// TwinCAT 3 PLC project MPLR
// ProgramVersion: 3.1.4026.19
// libraries:
//   Tc2_MC2, * (Beckhoff Automation GmbH)
//   Tc2_SerialCom, * (Beckhoff Automation GmbH)
//   Tc2_Standard, * (Beckhoff Automation GmbH)
//   Tc2_System, * (Beckhoff Automation GmbH)
//   Tc2_Utilities, * (Beckhoff Automation GmbH)
//   Tc3_Vision, * (Beckhoff Automation GmbH)
//   Tc3_Weighing, * (Beckhoff Automation GmbH)
// project tree:
//   DUTs/ E_PlateNum.TcDUT, MoveState_t.TcDUT, ST_CameraControl.TcDUT, ST_Origins.TcDUT, ST_PoseLREAL.TcDUT, ST_StepperMotorControl.TcDUT, ST_Transitions.TcDUT
//   DUTs/Robot/ur_input/ UR_1_T2O_Robot.TcDUT, UR_1_T2O_Safety.TcDUT, UR_1_T2O_State.TcDUT, UR_2_T2O_IO.TcDUT, UR_2_T2O_IOs.TcDUT, UR_2_T2O_Tool.TcDUT, UR_3_T2O_Joints.TcDUT, UR_4_T2O_TCP.TcDUT, UR_5_T2O_BitRegisters.TcDUT, UR_6_T2O_IntRegisters.TcDUT, UR_7_T2O_FloatRegisters.TcDUT, UR_T2O.TcDUT
//   DUTs/Robot/ur_output/ UR_8_O2T_IOs.TcDUT, UR_8_O2T_Robot.TcDUT, UR_8_O2T_Robot_IO.TcDUT, UR_9_O2T_Bits1.TcDUT, UR_9_O2T_Bits2.TcDUT, UR_9_O2T_Floats.TcDUT, UR_9_O2T_Ints.TcDUT, UR_9_O2T_Registers1.TcDUT, UR_9_O2T_Registers2.TcDUT, UR_O2T.TcDUT
//   GVLs/ process_gvl.TcGVL
//   / PlcTask.TcTTO
//   POUs/ FB_CreateTransformationMat.TcPOU, FB_LoadCell.TcPOU, FB_MagStirrer.TcPOU, FB_MatConversion.TcPOU, FB_MotorJog.TcPOU, FB_MultiplyMatrices4x4.TcPOU, FB_PeristalticPump.TcPOU, FB_Robot.TcPOU, FB_Camera.TcPOU, FB_SerialCom.TcPOU, FB_Test.TcPOU, MAIN.TcPOU, MPLR_UML.TcCD (not stored)
//   POUs/Modules/ FB_LoadingStationA.TcPOU, FB_SolidSamplingModule.TcPOU, FB_StirringModule.TcPOU
// real-time tasks:
//   TASK PlcTask: cycle T#10ms, priority 20, ADS port 350
//   TASK VnTask ImgAcq (Camera Daheng): cycle T#1ms, priority 5, ADS port 351
//   TASK VnTask ADS (Camera Daheng): cycle T#10ms, priority 6, ADS port 352
//   TASK VnTask ImgAcq (Daheng): cycle T#1ms, priority 7, ADS port 353
//   TASK VnTask ADS (Daheng): cycle T#10ms, priority 8, ADS port 354
//   TASK RTTask: cycle T#1ms, priority 1, ADS port 301
// motion (NC):
//   TASK NC-Task 1 SAF: cycle T#2ms, priority 4, ADS port 501
//   TASK NC-Task 1 SVB: cycle T#10ms, priority 9, ADS port 511
//   AXIS Axis 2 (id 2)
//     Dynamic: Acceleration=1314.17, Deceleration=1314.17, Jerk=3942.52
//     Velo: RefSearch=8.76116, RefSync=8.76116, SlowManual=43.8058, FastManual=262.8348, Fast=876.116, Maximum=876.116
//     PositionAreaControl: Enable=false
//     TargetPosControl: Enable=false
//     OtherSettings: AllowMotionCmdToSlave=true
//     encoder EncType=19
//       EncPara: ScaleFactorNumerator=60, ScaleFactorDenominator=1048576, MaxCount=#xffffffff
//         SoftEndMinControl: Range=5
//         SoftEndMaxControl: Range=17
//     drive DrvType=16
//       DrvPara: MaxCount=#xffffffff, DriveControlDWord=#x00020100
//         Analog: VeloReferenz=963.7276, VeloScale=32, TorqueSetpointScale=10, ScaleFactorActTorque=0.1
//         TimeComp: TaskDelayCycles=1
//     controller CtrType=1
//       CtrPara: PriorControlFactor=1
//         PosDiffControl: Enable=false
//         Observer: BandWidth=20
// I/O:
//   DEVICE Device 1 (EtherCAT), AmsNetId 5.146.234.225.2.1
//     Term 7 (EK1200) [EK1200-5000 EtherCAT Power supply (2A E-Bus)]
//       Term 7 (EL7062) [EL7062-0000 2Ch. Stepper motor output stage (48V, 3A)]
//         startup 32785:27 := 6C030000 // DRV Motor Settings Ch.1 / Motor speed limitation
//         startup 28688:3 := 08 // DRV Outputs Ch.1 / Modes of operation
//         startup 28688:16 := FF7F // DRV Outputs Ch.1 / Positive torque limit value
//         startup 28688:17 := FF7F // DRV Outputs Ch.1 / Negative torque limit value
//         startup 32784:87 := 64 // DRV Amplifier Settings Ch.1 / Position loop velocity feed forward gain
//         startup 32784:109 := 64000000 // DRV Amplifier Settings Ch.1 / Torque feed forward gain
//         startup 32785:52 := 70170000 // DRV Motor Settings Ch.1 / Configured motor current
//         startup 32784:19 := 1D00 // DRV Amplifier Settings Ch.1 / Current loop proportional gain
//         startup 32784:18 := 1E00 // DRV Amplifier Settings Ch.1 / Current loop integral time
//         startup 32784:21 := 91000000 // DRV Amplifier Settings Ch.1 / Velocity loop proportional gain
//         startup 32784:20 := 96000000 // DRV Amplifier Settings Ch.1 / Velocity loop integral time
//         startup 32776:18 := 0100 // FB Settings ENC Ch.1 / Encoder type
//         startup 32784:100 := 12 // DRV Amplifier Settings Ch.1 / Commutation type
//       Term 3 (EL1008) [EL1008 8Ch. Dig. Input 24V, 3ms]
//       Term 4 (EL3078) [EL3078 8Ch. Ana. Input +/-10V, +/-20mA]
//       Term 5 (EL2008) [EL2008 8Ch. Dig. Output 24V, 0.5A]
//       Term 12 (EL6002) [EL6002 Interface 2Ch. (RS232)]
//       Term 13 (EL9011) [EL9011 End Terminal]
//   DEVICE Device 3 (RT-Ethernet Adapter)
//   DEVICE Device 2 (Profinet Controller), AmsNetId 5.146.234.225.3.1
//     uriodev1 [Universal Robots A/S UR IO device, for PNIO controller with PDev 0000201]
//       modules: Term 1 (DAP Module), Term 2 (1_T2O State), Term 3 (2_T2O IO), Term 4 (3_T2O Joints), Term 5 (4_T2O TCP), Term 6 (5_T2O General Purpose Bit Registers), Term 7 (6_T2O General Purpose Int Registers), Term 8 (7_T2O General Purpose Float Registers), Term 9 (8_O2T Robot IO), Term 10 (9_O2T General Purpose Registers 1), Term 11 (10_O2T General Purpose Registers 2)
// variable links:
//   NC-Task 1 SAF/Axes/Axis 2 <-> Device 1 (EtherCAT)/Term 7 (EK1200)/Term 7 (EL7062)
//     Drive/Inputs/In/nDataIn1 <-> DRV Following error actual value Channel 1/Following error actual value
//     Drive/Inputs/In/nDcOutputTime <-> InfoData/DcOutputShift
//     Drive/Inputs/In/nState1 <-> DRV Statusword Channel 1/Statusword
//     Drive/Inputs/In/nState2 <-> DRV Statusword Channel 1/Statusword @bit 8
//     Drive/Inputs/In/nState4 @bit 1 <-> WcState/InputToggle
//     Drive/Inputs/In/nState4 <-> WcState/WcState
//     Drive/Outputs/Out/nCtrl1 <-> DRV Controlword Channel 1/Controlword
//     Drive/Outputs/Out/nCtrl2 <-> DRV Controlword Channel 1/Controlword @bit 8
//     Drive/Outputs/Out/nDataOut1 <-> DRV Target position Channel 1/Target position
//     Enc/Inputs/In/nDataIn1 <-> FB Position Channel 1/Position
//     Enc/Inputs/In/nDcInputTime <-> InfoData/DcInputShift
//     Enc/Inputs/In/nState4 @bit 1 <-> WcState/InputToggle
//     Enc/Inputs/In/nState4 <-> WcState/WcState
//   mplr/mplr Instance <-> Device 2 (Profinet Controller)/uriodev1
//     PlcTask Inputs/process_gvl.fRobotInput/General_Bits <-> API/Term 6 (5_T2O General Purpose Bit Registers)/Subterm 8 (5_T2O General Purpose Bit Registers)/Inputs/T2O Bit Registers
//     PlcTask Inputs/process_gvl.fRobotInput/General_Float/Floats <-> API/Term 8 (7_T2O General Purpose Float Registers)/Subterm 10 (7_T2O General Purpose Float Registers)/Inputs/T2O Float Registers
//     PlcTask Inputs/process_gvl.fRobotInput/General_Int/Ints <-> API/Term 7 (6_T2O General Purpose Int Registers)/Subterm 9 (6_T2O General Purpose Int Registers)/Inputs/T2O Int Registers
//     PlcTask Inputs/process_gvl.fRobotInput/IO <-> API/Term 3 (2_T2O IO)/Subterm 5 (2_T2O IO)/Inputs/T2O IO
//     PlcTask Inputs/process_gvl.fRobotInput/Joints <-> API/Term 4 (3_T2O Joints)/Subterm 6 (3_T2O Joints)/Inputs/T2O Joints
//     PlcTask Inputs/process_gvl.fRobotInput/State <-> API/Term 2 (1_T2O State)/Subterm 4 (1_T2O State)/Inputs/T2O State
//     PlcTask Inputs/process_gvl.fRobotInput/TCP <-> API/Term 5 (4_T2O TCP)/Subterm 7 (4_T2O TCP)/Inputs/T2O TCP
//     PlcTask Outputs/process_gvl.fRobotOutput/General_Register1 <-> API/Term 10 (9_O2T General Purpose Registers 1)/Subterm 12 (9_O2T General Purpose Registers 1)/Outputs/O2T Reg 1
//     PlcTask Outputs/process_gvl.fRobotOutput/General_Register2 <-> API/Term 11 (10_O2T General Purpose Registers 2)/Subterm 13 (10_O2T General Purpose Registers 2)/Outputs/O2T Reg 2
//     PlcTask Outputs/process_gvl.fRobotOutput/IO <-> API/Term 9 (8_O2T Robot IO)/Subterm 11 (8_O2T Robot IO)/Outputs/O2T IO
//   mplr/mplr Instance <-> NC-Task 1 SAF/Axes/Axis 2
//     PlcTask Inputs/MAIN.fbMotorJog.Axis1.NcToPlc <-> Outputs/ToPlc
//     PlcTask Outputs/MAIN.fbMotorJog.Axis1.PlcToNc <-> Inputs/FromPlc

CONFIGURATION MPLR
    RESOURCE PLC ON TwinCAT3
        TASK PlcTask(INTERVAL := T#10ms, PRIORITY := 20);
        PROGRAM MAIN WITH PlcTask : MAIN;
    END_RESOURCE
END_CONFIGURATION

// ---- DUTs/E_PlateNum.TcDUT
{attribute 'qualified_only'}
{attribute 'strict'}
{attribute 'to_string'}
TYPE E_PlateNum :
(
	ePlate1 := 0,
	ePlate2,
	ePlate3,
	ePlate4,
	ePlate5,
	ePlate6,
	ePlate7,
	ePlate8
);
END_TYPE

// ---- DUTs/MoveState_t.TcDUT
// {attribute 'qualified_only'}
// {attribute 'strict'}
// {attribute 'to_string'}
TYPE MoveState_t :
(
	MOVESTATE_INIT,
	MOVESTATE_ENABLE,
	MOVESTATE_IDLE,
	MOVESTATE_FORWARD,
	MOVESTATE_BACKWARDS,
	MOVESTATE_HALT,
	MOVESTATE_BACKWARDSSLOW,
	MOVESTATE_NEWTARGETPOSITION,
	MOVESTATE_ERROR,
	MOVESTATE_RESET
) UDINT;
END_TYPE

// ---- DUTs/Robot/ur_input/UR_1_T2O_Robot.TcDUT
TYPE UR_1_T2O_Robot :
STRUCT
	Controller_major_version:USINT;
	Controller_minor_version:USINT;
	Reserved:UInt;
	Robot_mode:USInt;
	Real_time_machine_seconds:USInt;
	Real_time_machine_milliseconds:UInt;
	Real_time_machine_minutes:USInt;
	Real_time_machine_hours:USInt;
	Real_time_machine_days:UINT;
	Robot_current_A:REAL;
	Is_power_on:BIT;
	Is_program_running:BIT;
	Is_teach_button_pressed:BIT;
	Is_power_button_pressed:BIT;
	Reserved_4:BIT;
	Reserved_5:BIT;
	Reserved_6:BIT;
	Reserved_7:BIT;
	Reserved_8_15:USInt;
	Reserved_16_31:UINT;
	Speed_slider_fraction:REAL;
END_STRUCT
END_TYPE

// ---- DUTs/Robot/ur_input/UR_1_T2O_Safety.TcDUT
TYPE UR_1_T2O_Safety :
STRUCT
	Safety_mode:USINT;
	Reserved_1:USINT;
	Reserved_2:UInt;
	Is_normal_mode:BIT;
	Is_reduced_mode:BIT;
	Is_protective_stopped:BIT;
	Is_recovery_mode:BIT;
	Is_safeguard_stopped:BIT;
	Is_system_emergency_stopped:BIT;
	Is_robot_emergency_stopped:BIT;
	Is_emergency_stopped:BIT;
	Is_violation:BIT;
	Is_fault:BIT;
	Is_stopped_due_to_safety:BIT;
	Reserved_11:BIT;
	Reserved_12:BIT;
	Reserved_13:BIT;
	Reserved_14:BIT;
	Reserved_15:BIT;
	Reserved_16_31:UINT;
END_STRUCT
END_TYPE

// ---- DUTs/Robot/ur_input/UR_1_T2O_State.TcDUT
TYPE UR_1_T2O_State :
STRUCT
      Robot : UR_1_T2O_Robot;
      Safety : UR_1_T2O_Safety;
END_STRUCT
END_TYPE

// ---- DUTs/Robot/ur_input/UR_2_T2O_IO.TcDUT
TYPE UR_2_T2O_IO :
STRUCT
	  IOs : UR_2_T2O_IOs;
	  Tool : UR_2_T2O_Tool;
END_STRUCT
END_TYPE

// ---- DUTs/Robot/ur_input/UR_2_T2O_IOs.TcDUT
TYPE UR_2_T2O_IOs :
STRUCT
	Standard_digital_inputs : USINT;
	Configurable_digital_inputs:USINT;
	Standard_digital_outputs:USINT;
	Configurable_digital_outputs:USINT;
	Analog_IO_types:USINT;
	Reserved_8_15:USINT;
	Reserved_16_31:UINT;
	Standard_analog_input_A_or_V:ARRAY[0..1] OF REAL;
	Standard_analog_output_A_or_V:ARRAY[0..1] OF REAL;
	IO_current_A:REAL;
	Euromap67_input_bits:ARRAY[0..3] OF BYTE;
	Euromap67_output_bits:ARRAY[0..3] OF BYTE;
	Euromap67_24V_voltage:REAL;
	Euromap67_24V_current:REAL;
END_STRUCT
END_TYPE

// ---- DUTs/Robot/ur_input/UR_2_T2O_Tool.TcDUT
TYPE UR_2_T2O_Tool :
STRUCT
	Tool_mode:USINT;
	Reserved_7_15:USINT;
	Reserved_16_31:UINT;
	Tool_Digital_Inputs:USINT;
	Tool_Digital_Outputs:USINT;
	Tool_Analog_Input_Types:USINT;
	Reserved_24_31:USINT;
	Tool_analog_input_A_OR_V:ARRAY[0..1] OF REAL;
	Tool_output_voltage_V:REAL;
	Tool_current_A:REAL;
END_STRUCT
END_TYPE

// ---- DUTs/Robot/ur_input/UR_3_T2O_Joints.TcDUT
TYPE UR_3_T2O_Joints :
STRUCT
	Joint_position_rad:ARRAY[0..5] OF REAL;
	Joint_velocity_radS:ARRAY[0..5] OF REAL;
	Joint_current_A:ARRAY[0..5] OF REAL;
	Joint_temperature_C:ARRAY[0..5] OF REAL;
	Joint_mode:ARRAY[0..5] OF USINT;
	Reserved_9:UINT;
END_STRUCT
END_TYPE

// ---- DUTs/Robot/ur_input/UR_4_T2O_TCP.TcDUT
TYPE UR_4_T2O_TCP :
STRUCT
	TCP_Position_XYZ_m:ARRAY[0..2] OF REAL;
	TCP_Position_RXRYRZ_rad:ARRAY[0..2] OF REAL;
	TCP_velocity_XYZ_m_S:ARRAY[0..2] OF REAL;
	TCP_velocity_RXRYRZ_rad_S:ARRAY[0..2] OF REAL;
	TCP_force_XYZ_N:ARRAY[0..2] OF REAL;
	TCP_torque_XYZ_Nm:ARRAY[0..2] OF REAL;
	TCP_force_scalar_N:REAL;
END_STRUCT
END_TYPE

// ---- DUTs/Robot/ur_input/UR_5_T2O_BitRegisters.TcDUT
TYPE UR_5_T2O_BitRegisters :
STRUCT
	GPBitIN_0 : BIT;
	GPBitIN_1 : BIT;
	GPBitIN_2 : BIT;
	GPBitIN_3 : BIT;
	GPBitIN_4 : BIT;
	GPBitIN_5 : BIT;
	GPBitIN_6 : BIT;
	GPBitIN_7 : BIT;
	GPBitIN_8 : BIT;
	GPBitIN_9 : BIT;
	GPBitIN_10 : BIT;
	GPBitIN_11 : BIT;
	GPBitIN_12 : BIT;
	GPBitIN_13 : BIT;
	GPBitIN_14 : BIT;
	GPBitIN_15 : BIT;
	GPBitIN_16 : BIT;
	GPBitIN_17 : BIT;
	GPBitIN_18 : BIT;
	GPBitIN_19 : BIT;
	GPBitIN_20 : BIT;
	GPBitIN_21 : BIT;
	GPBitIN_22 : BIT;
	GPBitIN_23 : BIT;
	GPBitIN_24 : BIT;
	GPBitIN_25 : BIT;
	GPBitIN_26 : BIT;
	GPBitIN_27 : BIT;
	GPBitIN_28 : BIT;
	GPBitIN_29 : BIT;
	GPBitIN_30 : BIT;
	GPBitIN_31 : BIT;
	GPBitIN_32 : BIT;
	GPBitIN_33 : BIT;
	GPBitIN_34 : BIT;
	GPBitIN_35 : BIT;
	GPBitIN_36 : BIT;
	GPBitIN_37 : BIT;
	GPBitIN_38 : BIT;
	GPBitIN_39 : BIT;
	GPBitIN_40 : BIT;
	GPBitIN_41 : BIT;
	GPBitIN_42 : BIT;
	GPBitIN_43 : BIT;
	GPBitIN_44 : BIT;
	GPBitIN_45 : BIT;
	GPBitIN_46 : BIT;
	GPBitIN_47 : BIT;
	GPBitIN_48 : BIT;
	GPBitIN_49 : BIT;
	GPBitIN_50 : BIT;
	GPBitIN_51 : BIT;
	GPBitIN_52 : BIT;
	GPBitIN_53 : BIT;
	GPBitIN_54 : BIT;
	GPBitIN_55 : BIT;
	GPBitIN_56 : BIT;
	GPBitIN_57 : BIT;
	GPBitIN_58 : BIT;
	GPBitIN_59 : BIT;
	GPBitIN_60 : BIT;
	GPBitIN_61 : BIT;
	GPBitIN_62 : BIT;
	GPBitIN_63 : BIT;
END_STRUCT
END_TYPE

// ---- DUTs/Robot/ur_input/UR_6_T2O_IntRegisters.TcDUT
TYPE UR_6_T2O_IntRegisters :
STRUCT
		Ints:ARRAY[0..23] OF DINT;
END_STRUCT
END_TYPE

// ---- DUTs/Robot/ur_input/UR_7_T2O_FloatRegisters.TcDUT
TYPE UR_7_T2O_FloatRegisters :
STRUCT
	  Floats : ARRAY[0..23] OF REAL;
END_STRUCT
END_TYPE

// ---- DUTs/Robot/ur_input/UR_T2O.TcDUT
TYPE UR_T2O :
STRUCT
	State:UR_1_T2O_State;
	IO:UR_2_T2O_IO;
	Joints:UR_3_T2O_Joints;
	TCP:UR_4_T2O_TCP;
	General_Bits:UR_5_T2O_BitRegisters;
	General_Int:UR_6_T2O_IntRegisters;
	General_Float:UR_7_T2O_FloatRegisters;
END_STRUCT
END_TYPE

// ---- DUTs/Robot/ur_output/UR_8_O2T_IOs.TcDUT
TYPE UR_8_O2T_IOs :
STRUCT
	Standard_digital_output_mask:USINT;
	Configurable_digital_output_mask:USINT;
	Standard_digital_outputs:USINT;
	Configurable_digital_outputs:USINT;
	Analog_output_mask:USINT;
	Analog_output_types:USINT;
	Tool_digital_output_mask:USINT;
	Tool_digital_output:USINT;
	Standard_analog_output:ARRAY[0..1] OF REAL;
END_STRUCT
END_TYPE

// ---- DUTs/Robot/ur_output/UR_8_O2T_Robot.TcDUT
TYPE UR_8_O2T_Robot :
STRUCT
	  Speed_slider_fraction_mask : BIT;
	  Reserved_1 : BIT;
	  Reserved_2 : BIT;
	  Reserved_3 : BIT;
	  Reserved_4 : BIT;
	  Reserved_5 : BIT;
	  Reserved_6 : BIT;
	  Reserved_7 : BIT;
	  Reserved_8_15 : USINT;
	  Reserved_16_31 : UINT;
	  Speed_slider_fraction : REAL;
END_STRUCT
END_TYPE

// ---- DUTs/Robot/ur_output/UR_8_O2T_Robot_IO.TcDUT
TYPE UR_8_O2T_Robot_IO :
STRUCT
      Robot : UR_8_O2T_Robot;
      IOs : UR_8_O2T_IOs;
END_STRUCT
END_TYPE

// ---- DUTs/Robot/ur_output/UR_9_O2T_Bits1.TcDUT
TYPE UR_9_O2T_Bits1 :
STRUCT
	GPBitIN_0 : BIT;
	GPBitIN_1 : BIT;
	GPBitIN_2 : BIT;
	GPBitIN_3 : BIT;
	GPBitIN_4 : BIT;
	GPBitIN_5 : BIT;
	GPBitIN_6 : BIT;
	GPBitIN_7 : BIT;
	GPBitIN_8 : BIT;
	GPBitIN_9 : BIT;
	GPBitIN_10 : BIT;
	GPBitIN_11 : BIT;
	GPBitIN_12 : BIT;
	GPBitIN_13 : BIT;
	GPBitIN_14 : BIT;
	GPBitIN_15 : BIT;
	GPBitIN_16 : BIT;
	GPBitIN_17 : BIT;
	GPBitIN_18 : BIT;
	GPBitIN_19 : BIT;
	GPBitIN_20 : BIT;
	GPBitIN_21 : BIT;
	GPBitIN_22 : BIT;
	GPBitIN_23 : BIT;
	GPBitIN_24 : BIT;
	GPBitIN_25 : BIT;
	GPBitIN_26 : BIT;
	GPBitIN_27 : BIT;
	GPBitIN_28 : BIT;
	GPBitIN_29 : BIT;
	GPBitIN_30 : BIT;
	GPBitIN_31 : BIT;
END_STRUCT
END_TYPE

// ---- DUTs/Robot/ur_output/UR_9_O2T_Bits2.TcDUT
TYPE UR_9_O2T_Bits2 :
STRUCT
	GPBitIN_32 : BIT;
	GPBitIN_33 : BIT;
	GPBitIN_34 : BIT;
	GPBitIN_35 : BIT;
	GPBitIN_36 : BIT;
	GPBitIN_37 : BIT;
	GPBitIN_38 : BIT;
	GPBitIN_39 : BIT;
	GPBitIN_40 : BIT;
	GPBitIN_41 : BIT;
	GPBitIN_42 : BIT;
	GPBitIN_43 : BIT;
	GPBitIN_44 : BIT;
	GPBitIN_45 : BIT;
	GPBitIN_46 : BIT;
	GPBitIN_47 : BIT;
	GPBitIN_48 : BIT;
	GPBitIN_49 : BIT;
	GPBitIN_50 : BIT;
	GPBitIN_51 : BIT;
	GPBitIN_52 : BIT;
	GPBitIN_53 : BIT;
	GPBitIN_54 : BIT;
	GPBitIN_55 : BIT;
	GPBitIN_56 : BIT;
	GPBitIN_57 : BIT;
	GPBitIN_58 : BIT;
	GPBitIN_59 : BIT;
	GPBitIN_60 : BIT;
	GPBitIN_61 : BIT;
	GPBitIN_62 : BIT;
	GPBitIN_63 : BIT;
END_STRUCT
END_TYPE

// ---- DUTs/Robot/ur_output/UR_9_O2T_Floats.TcDUT
TYPE UR_9_O2T_Floats :
STRUCT
	Floats : ARRAY[0..11] OF REAL;
END_STRUCT
END_TYPE

// ---- DUTs/Robot/ur_output/UR_9_O2T_Ints.TcDUT
TYPE UR_9_O2T_Ints :
STRUCT
      Ints : ARRAY[0..11] OF DINT;
END_STRUCT
END_TYPE

// ---- DUTs/Robot/ur_output/UR_9_O2T_Registers1.TcDUT
TYPE UR_9_O2T_Registers1 :
STRUCT
      Bits : UR_9_O2T_Bits1;
      Ints : UR_9_O2T_Ints;
      Floats : UR_9_O2T_Floats;
END_STRUCT
END_TYPE

// ---- DUTs/Robot/ur_output/UR_9_O2T_Registers2.TcDUT
TYPE UR_9_O2T_Registers2 :
STRUCT
      Bits : UR_9_O2T_Bits2;
      Ints : UR_9_O2T_Ints;
      Floats : UR_9_O2T_Floats;
END_STRUCT
END_TYPE

// ---- DUTs/Robot/ur_output/UR_O2T.TcDUT
TYPE UR_O2T :
STRUCT
	IO:UR_8_O2T_Robot_IO;
	General_Register1:UR_9_O2T_Registers1;
	General_Register2:UR_9_O2T_Registers1;
END_STRUCT
END_TYPE

// ---- DUTs/ST_CameraControl.TcDUT
TYPE ST_CameraControl :
STRUCT

END_STRUCT
END_TYPE

// ---- DUTs/ST_Origins.TcDUT
TYPE ST_Origins :
STRUCT
	fOrigin1		: ARRAY[0..5]	OF LREAL := [0.0, 0.0, 0.0, 0.0, 0.0, 0.0];
	fOrigin2		: ARRAY[0..5]	OF LREAL := [0.0, 0.0, 0.0, 0.0, 0.0, 0.0];
	fOrigin3		: ARRAY[0..5]	OF LREAL := [0.0, 0.0, 0.0, 0.0, 0.0, 0.0];
	fOrigin4		: ARRAY[0..5]	OF LREAL := [0.0, 0.0, 0.0, 0.0, 0.0, 0.0];
	fOrigin5		: ARRAY[0..5]	OF LREAL := [0.0, 0.0, 0.0, 0.0, 0.0, 0.0];
	fOrigin6		: ARRAY[0..5]	OF LREAL := [0.0, 0.0, 0.0, 0.0, 0.0, 0.0];
	fOrigin7		: ARRAY[0..5]	OF LREAL := [0.0, 0.0, 0.0, 0.0, 0.0, 0.0];
	fOrigin8		: ARRAY[0..5]	OF LREAL := [0.0, 0.0, 0.0, 0.0, 0.0, 0.0];
END_STRUCT
END_TYPE

// ---- DUTs/ST_PoseLREAL.TcDUT
TYPE ST_PoseLREAL :
STRUCT
	R_Mat : TcVnMatrix3x3_LREAL;
    T_Mat : TcVnVector3_LREAL;
	X_Mat : TcVnMatrix;
END_STRUCT
END_TYPE

// ---- DUTs/ST_StepperMotorControl.TcDUT
TYPE ST_StepperMotorControl :
STRUCT
// 	Axis1:AXIS_REF;
// 	MC_Power: MC_Power;
// 	MC_MoveAbsolute: MC_MoveAbsolute;
// 	bMove: BOOL;
// 	bInput AT%I*:BOOL;
// 	bEnable: BOOL;
// 	
// 	bLoadingPosition		:LREAL	:=68;
// 	bLoadingVelocity		:LREAL	:=0.5;
// 	bLoadingAcceleration	:LREAL	:=1;
// 	bLoadingDeceleration	:LREAL	:=1;
// 	
// 	bDosingPosition		:LREAL	:=64;
// 	bDosingVelocity		:LREAL	:=0.5;
// 	bDosingAcceleration	:LREAL	:=1;
// 	bDosingDeceleration	:LREAL	:=1;
END_STRUCT
END_TYPE

// ---- DUTs/ST_Transitions.TcDUT
TYPE ST_Transitions :
STRUCT
	ModulesDetected				: BOOL;
	FlaskPicked					: BOOL;
	FlaskPlaced					: BOOL;
	FingerAGripped				: BOOL;
	FingerBGripped				: BOOL;
	FingerCGripped				: BOOL;
	FingerDGripped				: BOOL;
	FingerADeGripped			: BOOL;
	FingerBDeGripped			: BOOL;
	FingerCDeGripped			: BOOL;
	FingerDDeGripped			: BOOL;
	DosedTargetWeight			: BOOL;
	InputBottleDecapped			: BOOL;
	DetectedPlates				: BOOL;		// QR code triggered and Plates detected
	MotorInPos					: BOOL;		
	
	TabletsPoured				: BOOL;
	VibrationDone				: BOOL;
	TabletsDetected				: BOOL;
	InputBottlePlaced			: BOOL;
	TabletPicked				: BOOL;
	TabletRebottled				: BOOL;
	InputBottleCapped			: BOOL;
	InputBottleRemoved			: BOOL;
	OutputBottleTransferred 	: BOOL;
	OutputBottleDecapped		: BOOL;
	CameraParamsChanged			: BOOL;
	ImprintDetectionPoseReached	: BOOL;
	ImprintCheckDone			: BOOL;
	ImprintRecheckDone			: BOOL;
	TabletFlipped				: BOOL;
	TabletLoaded				: BOOL;
	MatrixLoaded				: BOOL;
	MeasurementDone				: BOOL;
	MatrixUnloaded				: BOOL;
	TabletUnloaded				: BOOL;
	OutputBottleCapped 			: BOOL;
	OutputBottleRemoved			: BOOL;
	SampleRemoved				: BOOL;
	SystemReset					: BOOL;
END_STRUCT
END_TYPE

// ---- GVLs/process_gvl.TcGVL
{attribute 'qualified_only'}
VAR_GLOBAL
	fRobotInput		AT%I*:	UR_T2O;		(* Outputs from Robot to PLC *)
	fRobotOutput	AT%Q*:	UR_O2T;		(* Inputs from PLC to Robot *)
// 	fMotorControl		:	ST_StepperMotorControl;
	fCameraControl		:	ST_CameraControl;	
	RxBufferEL			: ComBuffer;	(* Receive data buffer; used with all receive function blocks *)
	TxBufferEL			: ComBuffer;
//	Plate information
END_VAR

// ---- POUs/MAIN.TcPOU
PROGRAM MAIN
VAR
	fbRobot			:	FB_Robot;
	fbMotorJog		:	FB_MotorJog;
	fbCamera		:	FB_Camera;
	stTransitions	:	ST_Transitions;
	bStartProcess	:	BOOL := TRUE;
	
// 	TaskId			: process_gvl.fRobotOutput.General_Register1.Ints.Ints[0];
	
	bMove : BOOL;
	nIdlePosition : INT := 1;
	bFlag : BOOL := FALSE;
END_VAR

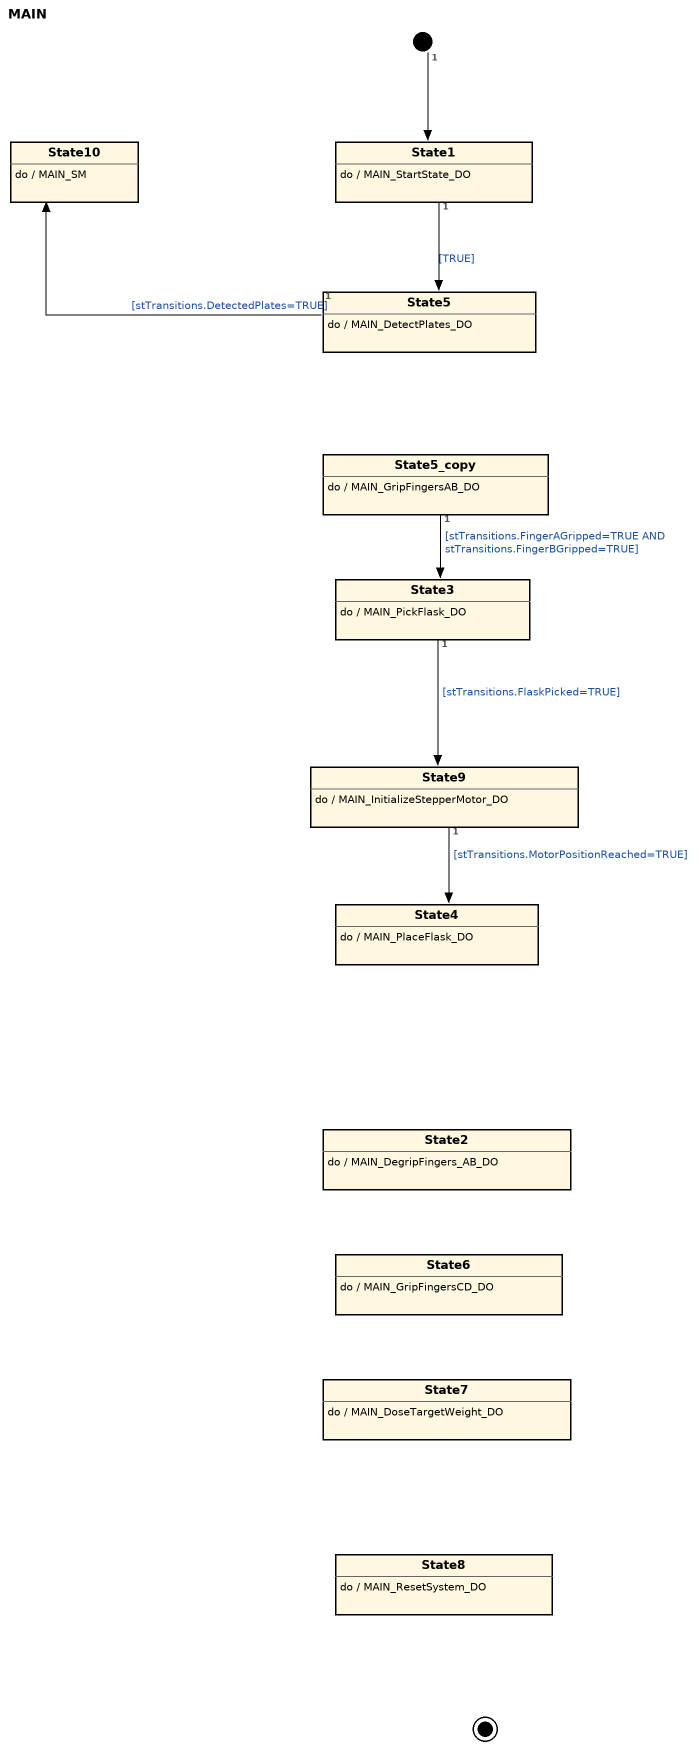
STATECHART MAIN  // abortable
    START StartState1
    STATE State10
        do / MAIN_SM
    STATE State1
        do / MAIN_StartState_DO
    STATE State5
        do / MAIN_DetectPlates_DO
    STATE State5_copy
        do / MAIN_GripFingersAB_DO
    STATE State3
        do / MAIN_PickFlask_DO
    STATE State9
        do / MAIN_InitializeStepperMotor_DO
    STATE State4
        do / MAIN_PlaceFlask_DO
    STATE State2
        do / MAIN_DegripFingers_AB_DO
    STATE State6
        do / MAIN_GripFingersCD_DO
    STATE State7
        do / MAIN_DoseTargetWeight_DO
    STATE State8
        do / MAIN_ResetSystem_DO
    END EndState1
    StartState1 -> State1  // priority 1, on completion
    State1 -> State5 [TRUE] // priority 1
    State5 -> State10 [stTransitions.DetectedPlates=TRUE] // priority 1
    State5_copy -> State3 [stTransitions.FingerAGripped=TRUE AND stTransitions.FingerBGripped=TRUE] // priority 1
    State3 -> State9 [stTransitions.FlaskPicked=TRUE] // priority 1
    State9 -> State4 [stTransitions.MotorPositionReached=TRUE] // priority 1
END_STATECHART

ACTION MAIN_DegripFingers_AB_DO:

IF stTransitions.DosedTargetWeight THEN
	stTransitions.FingerADeGripped := fbRobot.DeGripFingerA();
END_IF
IF stTransitions.FingerAGripped THEN
	stTransitions.FingerBDeGripped := fbRobot.DeGripFingerB();
// 	fbRobot.SendTaskId(0); 
END_IF
END_ACTION

ACTION MAIN_DegripFingers_CD_DO:

END_ACTION

ACTION MAIN_DetectPlates_DO:
// Initialize camera and detect QR codes
// stTransitions.DetectedPlates := fbCamera.QRCodefinal();

stTransitions.DetectedPlates := bFlag;
// Start UR TP program for detection of QR codes
// Write data to robot
END_ACTION

ACTION MAIN_DoseTargetWeight_DO:

END_ACTION

ACTION MAIN_GripFingersAB_DO:
(* Program for Gripping Fingers on Deposit station AB *)

// Reset previous transition states

// Run Program on TP
IF bStartProcess THEN
	stTransitions.FingerAGripped := fbRobot.GripFingerA();
END_IF
IF stTransitions.FingerAGripped THEN
	stTransitions.FingerBGripped := fbRobot.GripFingerB();
// 	fbRobot.SendTaskId(0);
END_IF
END_ACTION

ACTION MAIN_GripFingersCD_DO:

END_ACTION

ACTION MAIN_InitializeStepperMotor_DO:
// Stepper motor initialization

// fbMotorJog.EnablePower();
// fbMotorJog.MotorLoadingPosition();
// fbMotorJog.MotorDosingPosition();

// Find out flag for target reaching of stepper motor
END_ACTION

ACTION MAIN_PickFlask_DO:
// Trigger Pick and place of Flask from Input Application plate

// fbRobot.SendTaskId(xx);
stTransitions.FlaskPicked	:= fbRobot.PickFlask();
END_ACTION

ACTION MAIN_PlaceFlask_DO:
// fbRobot.SendTaskId(xx);

// reset previous transitions
stTransitions.MotorPositionReached:=FALSE;

//
END_ACTION

ACTION MAIN_ResetSystem_DO:

END_ACTION

ACTION MAIN_SM:
fbMotorJog.MotorMove(bMove, nIdlePosition);
END_ACTION

ACTION MAIN_StartState_DO:
// Variables Initializations

// fbMotorJog.EnablePower();
// fbMotorJog.MotorDosingPosition();

// Inputs from Robot to PLC

// Visualization button for bStartProcess manual trigger
END_ACTION

END_PROGRAM

// ---- POUs/FB_Robot.TcPOU
FUNCTION_BLOCK FB_Robot
VAR_INPUT
END_VAR
VAR_OUTPUT
	r1_matrix       : TcVnMatrix3x3_LREAL;
	v1_matrix 		: TcVnVector3_LREAL;
END_VAR
VAR
	_TCPPoseT : ARRAY[0..2] OF LREAL := [1.0, 1.0, 1.0];
	fb_Convert_1 : FB_MatConversion;
	
	fbmakeT1 : FB_CreateTransformationMat; 
	T4x4_matrix_1       : TcVnMatrix;
END_VAR

METHOD DeGripFingerA : BOOL
VAR_INPUT
END_VAR

VAR
	bTaskStatus : BOOL := FALSE; //
END_VAR
SendTaskId(30);

bTaskStatus := process_gvl.fRobotInput.General_Bits.GPBitIN_35;

IF bTaskStatus THEN
	DeGripFingerA := TRUE;
	SendTaskId(0); 
END_IF
END_METHOD

METHOD DeGripFingerB : BOOL
VAR_INPUT
END_VAR

VAR
	bTaskStatus : BOOL := FALSE; //
END_VAR
SendTaskId(40);

bTaskStatus := process_gvl.fRobotInput.General_Bits.GPBitIN_35;

IF bTaskStatus THEN
	DeGripFingerB := TRUE;
	SendTaskId(0); 
END_IF
END_METHOD

METHOD DeGripFingerC : BOOL
VAR_INPUT
END_VAR

VAR
	bTaskStatus : BOOL := FALSE; //
END_VAR
SendTaskId(7);

bTaskStatus := process_gvl.fRobotInput.General_Bits.GPBitIN_35;

IF bTaskStatus THEN
	DeGripFingerC := TRUE;
	SendTaskId(0); 
END_IF
END_METHOD

METHOD DeGripFingerD : BOOL
VAR_INPUT
END_VAR

VAR
	bTaskStatus : BOOL := FALSE; //
END_VAR
SendTaskId(7);

bTaskStatus := process_gvl.fRobotInput.General_Bits.GPBitIN_35;

IF bTaskStatus THEN
	DeGripFingerD := TRUE;
	SendTaskId(0); 
END_IF
END_METHOD

METHOD DeGripFingerE : BOOL
VAR_INPUT
END_VAR

VAR
	bTaskStatus : BOOL := FALSE; //
END_VAR
SendTaskId(7);

bTaskStatus := process_gvl.fRobotInput.General_Bits.GPBitIN_35;

IF bTaskStatus THEN
	DeGripFingerE := TRUE;
	SendTaskId(0); 
END_IF
END_METHOD

METHOD DeGripFingerF : BOOL
VAR_INPUT
END_VAR

VAR
	bTaskStatus : BOOL := FALSE; //
END_VAR
SendTaskId(7);

bTaskStatus := process_gvl.fRobotInput.General_Bits.GPBitIN_35;

IF bTaskStatus THEN
	DeGripFingerF := TRUE;
	SendTaskId(0); 
END_IF
END_METHOD

METHOD GripFingerA : BOOL
VAR_INPUT
END_VAR

VAR
	bTaskStatus : BOOL := FALSE; //
END_VAR
SendTaskId(10);

bTaskStatus := process_gvl.fRobotInput.General_Bits.GPBitIN_35;

IF bTaskStatus THEN
	GripFingerA := TRUE;
	SendTaskId(0); 
END_IF
END_METHOD

METHOD GripFingerB : BOOL
VAR_INPUT
END_VAR

VAR
	bTaskStatus : BOOL := FALSE; //
END_VAR
SendTaskId(20);

bTaskStatus := process_gvl.fRobotInput.General_Bits.GPBitIN_35;

IF bTaskStatus THEN
	GripFingerB := TRUE;
	SendTaskId(0); 
END_IF
END_METHOD

METHOD GripFingerC : BOOL
VAR_INPUT
END_VAR

VAR
	bTaskStatus : BOOL := FALSE; //
END_VAR
SendTaskId(7);

bTaskStatus := process_gvl.fRobotInput.General_Bits.GPBitIN_35;

IF bTaskStatus THEN
	GripFingerC := TRUE;
	SendTaskId(0); 
END_IF
END_METHOD

METHOD GripFingerD : BOOL
VAR_INPUT
END_VAR

VAR
	bTaskStatus : BOOL := FALSE; //
END_VAR
SendTaskId(7);

bTaskStatus := process_gvl.fRobotInput.General_Bits.GPBitIN_35;

IF bTaskStatus THEN
	GripFingerD := TRUE;
	SendTaskId(0); 
END_IF
END_METHOD

METHOD GripFingerE : BOOL
VAR_INPUT
END_VAR

VAR
	bTaskStatus : BOOL := FALSE; //
END_VAR
SendTaskId(7);

bTaskStatus := process_gvl.fRobotInput.General_Bits.GPBitIN_35;

IF bTaskStatus THEN
	GripFingerE := TRUE;
	SendTaskId(0); 
END_IF
END_METHOD

METHOD GripFingerF : BOOL
VAR_INPUT
END_VAR

VAR
	bTaskStatus : BOOL := FALSE; //
END_VAR
SendTaskId(7);

bTaskStatus := process_gvl.fRobotInput.General_Bits.GPBitIN_35;

IF bTaskStatus THEN
	GripFingerF := TRUE;
	SendTaskId(0); 
END_IF
END_METHOD

METHOD Move_Home : BOOL
VAR_INPUT
END_VAR

VAR
	bTaskStatus : BOOL := FALSE; //
END_VAR
SendTaskId(1);

bTaskStatus := process_gvl.fRobotInput.General_Bits.GPBitIN_35;		//WHat is this for?

IF bTaskStatus THEN
	Move_Home := TRUE;
	SendTaskId(0); 
END_IF
END_METHOD

METHOD PickFlask : BOOL
VAR_INPUT
END_VAR

VAR
	bTaskStatus : BOOL := FALSE; //
END_VAR
SendTaskId(7);

bTaskStatus := process_gvl.fRobotInput.General_Bits.GPBitIN_35;

IF bTaskStatus THEN
	PickFlask := TRUE;
	SendTaskId(0); 
END_IF
END_METHOD

METHOD PlaceFlask : BOOL
VAR_INPUT
END_VAR

VAR
	bTaskStatus: BOOL := FALSE;
END_VAR
SendTaskId(7);

bTaskStatus := process_gvl.fRobotInput.General_Bits.GPBitIN_35;		// Define the GPBitIN_xx number for respective task number on TP 

IF bTaskStatus THEN
	PlaceFlask := TRUE;
	SendTaskId(0); 
END_IF
END_METHOD

METHOD RobotPose : TcVnMatrix
VAR_INPUT
END_VAR
VAR
	pose_x : REAL;
	pose_y : REAL;
	pose_z : REAL;
	pose_rx: REAL;
	pose_ry: REAL;
	pose_rz: REAL;
	Tpose_mat : ARRAY[0..3, 0..3] OF LREAL;
END_VAR
// pose_x:= 1000*LREAL_TO_REAL(process_gvl.fRobotInput.TCP.TCP_Position_XYZ_m[0]);
// pose_y:= 1000*LREAL_TO_REAL(process_gvl.fRobotInput.TCP.TCP_Position_XYZ_m[1]);
// pose_z:= 1000*LREAL_TO_REAL(process_gvl.fRobotInput.TCP.TCP_Position_XYZ_m[2]);
// pose_rx:=process_gvl.fRobotInput.TCP.TCP_Position_RXRYRZ_rad[0];
// pose_ry:=process_gvl.fRobotInput.TCP.TCP_Position_RXRYRZ_rad[1];
// pose_rz:=process_gvl.fRobotInput.TCP.TCP_Position_RXRYRZ_rad[2];

	pose_x := 0.1;
	pose_y := 0.1;
	pose_z := 0.1;
	pose_rx:= 0.1;
	pose_ry:= 0.1;
	pose_rz:= 0.1;

r1_matrix := fb_Convert_1.RotVecToRmat(rx:= pose_rx, ry:= pose_ry, rz:=pose_rz);
v1_matrix := fb_Convert_1.Make3x3Vec(pose_x, pose_y, pose_z);
// fbmakeT1.R_mat := r1_matrix;
// fbmakeT1.T_mat := v1_matrix;
// fbmakeT1();
// // T4x4_robotpose:=fbmakeT1.Tx_mat;
// RobotPose := fbmakeT1.Tx_mat;
// // RobotTCPPose REF= _TCPPoseT;
// // ---- publish as TcVnMatrix (header) ----
// // T4x4_robotpose.nRows := 4;
// // T4x4_robotpose.nCols := 4;
// // T4x4_robotpose.eType := TCVN_ET_LREAL;        // element type = LREAL (per ETcVnElementType)
// // T4x4_robotpose.pData := ADR(Tpose_mat);           // pointer to backing storage
END_METHOD

METHOD SendTaskId
VAR_INPUT
	nTaskId : INT;
END_VAR
process_gvl.fRobotOutput.General_Register1.Ints.Ints[0] := nTaskId;
END_METHOD

END_FUNCTION_BLOCK

// ---- POUs/FB_MatConversion.TcPOU
FUNCTION_BLOCK FB_MatConversion
VAR_INPUT
END_VAR
VAR_OUTPUT
END_VAR
VAR
END_VAR

METHOD Make3x3Vec : TcVnVector3_LREAL
VAR_INPUT
	x : LREAL;
    y : LREAL;
    z : LREAL;
END_VAR
VAR
    v : TcVnVector3_LREAL;
END_VAR

v[0] := x;
v[1] := y;
v[2] := z;

Make3x3Vec := v;
END_METHOD

METHOD RmatToRotVec : TcVnVector3_LREAL
VAR_INPUT
	    Rot : TcVnMatrix3x3_LREAL;
END_VAR
VAR
    tr, cosT, theta, s_a : LREAL;
    v 		: TcVnVector3_LREAL;
END_VAR
tr   := Rot[0,0] + Rot[1,1] + Rot[2,2];
cosT := (tr - 1.0) * 0.5;
IF cosT > 1.0 THEN
	cosT := 1.0;
END_IF
IF cosT < -1.0 THEN 
	cosT := -1.0; 
END_IF

theta := ACOS(cosT);
IF ABS(theta) < 1e-6 THEN
    v[0] := 0; v[1] := 0; v[2] := 0;
ELSE
    s_a := 1.0 / (2.0 * SIN(theta) + 1E-12);
    v[0] := (Rot[2,1] - Rot[1,2]) * s_a * theta;
    v[1] := (Rot[0,2] - Rot[2,0]) * s_a * theta;
    v[2] := (Rot[1,0] - Rot[0,1]) * s_a * theta;
END_IF


RmatToRotVec := v;
END_METHOD

METHOD RotVecToRmat : TcVnMatrix3x3_LREAL
VAR_INPUT
	rx : LREAL;   // roll  about X (rad)
    ry : LREAL;   // pitch about Y (rad)
    rz : LREAL;   // yaw   about Z (rad)
END_VAR
VAR_OUTPUT
    R_mat  : TcVnMatrix3x3_LREAL;  // Rotation matrix (Rz*Ry*Rx)
END_VAR
VAR
    cX, sX, cY, sY, cZ, sZ : LREAL;
END_VAR
// Compute once per call/scan
cX := COS(rx);  sX := SIN(rx);
cY := COS(ry);  sY := SIN(ry);
cZ := COS(rz);  sZ := SIN(rz);

// ZYX convention: R = Rz * Ry * Rx
R_mat[0,0] :=  cZ*cY;              R_mat[0,1] :=  cZ*sY*sX - sZ*cX;   R_mat[0,2] :=  cZ*sY*cX + sZ*sX;
R_mat[1,0] :=  sZ*cY;              R_mat[1,1] :=  sZ*sY*sX + cZ*cX;   R_mat[1,2] :=  sZ*sY*cX - cZ*sX;
R_mat[2,0] := -sY;                 R_mat[2,1] :=  cY*sX;              R_mat[2,2] :=  cY*cX;
END_METHOD

END_FUNCTION_BLOCK

// ---- POUs/FB_CreateTransformationMat.TcPOU
FUNCTION_BLOCK FB_CreateTransformationMat
VAR_INPUT
	R_mat : TcVnMatrix3x3_LREAL;   // rotation
    T_mat : TcVnVector3_LREAL;     // translation 
END_VAR
VAR_OUTPUT
	Tx_mat : TcVnMatrix;            // generic Vision matrix header
	Tr_mat : ARRAY[0..3, 0..3] OF LREAL;	
END_VAR
VAR

END_VAR

// Top-left 3x3 = R
Tr_mat[0,0] := R_mat[0,0];  Tr_mat[0,1] := R_mat[0,1];  Tr_mat[0,2] := R_mat[0,2];
Tr_mat[1,0] := R_mat[1,0];  Tr_mat[1,1] := R_mat[1,1];  Tr_mat[1,2] := R_mat[1,2];
Tr_mat[2,0] := R_mat[2,0];  Tr_mat[2,1] := R_mat[2,1];  Tr_mat[2,2] := R_mat[2,2];

// Right column = t
Tr_mat[0,3] := T_mat[0];
Tr_mat[1,3] := T_mat[1];
Tr_mat[2,3] := T_mat[2];

// Bottom row = [0 0 0 1]
Tr_mat[3,0] := 0.0;     
Tr_mat[3,1] := 0.0;     
Tr_mat[3,2] := 0.0;     
Tr_mat[3,3] := 1.0;

// ---- publish as TcVnMatrix (header) ----
Tx_mat.nRows := 4;
Tx_mat.nCols := 4;
Tx_mat.eType := TCVN_ET_LREAL;        // element type = LREAL (per ETcVnElementType)
Tx_mat.pData := ADR(Tr_mat);           // pointer to backing storage

END_FUNCTION_BLOCK

// ---- POUs/FB_MotorJog.TcPOU
FUNCTION_BLOCK FB_MotorJog EXTENDS FB_SolidSamplingModule
VAR_INPUT
END_VAR
VAR_OUTPUT
END_VAR
VAR
	
	/// axis reference data structure 
	Axis1: AXIS_REF;
	/// state machine state 
	state: MoveState_t;
	PowerAxis1: MC_Power;
	/// debug function block output data 
	PowerAxis1Out: ST_McOutputs;
	MoveAxis1: MC_MoveAbsolute;
	/// debug function block output data 
	MoveAbsoluteOut1: ST_McOutputs;
// 	MoveAxis2: MC_MoveAbsolute;
	/// debug function block output data 
// 	MoveAbsoluteOut2: ST_McOutputs;
	Reset: MC_Reset;
	/// debug function block output data 
	ResetOut: ST_McOutputs;
	
	HaltAxis1: MC_Halt;
	fbRobot		: FB_Robot;
	fbRise		: R_TRIG;
	bPulse		: BOOL;
	bEnable	:	BOOL := FALSE;
END_VAR

METHOD EnablePower : BOOL
VAR
END_VAR
Axis1.ReadStatus();

PowerAxis1(
	Axis:=Axis1, 
	Enable:= bEnable, 
	Status=> , 
	Busy=> , 
	Active=> , 
	Error=> , 
	ErrorID=> );
END_METHOD

METHOD MotorDosingPosition : BOOL
VAR_INPUT
END_VAR
END_METHOD

METHOD MotorLoadingPosition : BOOL
VAR_INPUT
END_VAR
END_METHOD

METHOD MotorMain : BOOL
VAR_INPUT
	bMove : BOOL;
	nIdlePosition : INT; // 1: 63, 2: 70
END_VAR
MotorMove(bMove, nIdlePosition);
RETURN;

IF nIdlePosition < 1 OR nIdlePosition > 2 THEN		// Rejects other Position values
	nIdlePosition := 1;
END_IF

	(* update the axis status at the beginning of each cycle *)
	Axis1();

	(* move axis using a state machine *)
	CASE state OF

		MOVESTATE_INIT :	(* initialisation *)
			MoveAxis1.Execute := FALSE;
			Reset.Execute := FALSE;
			state := MOVESTATE_ENABLE;

		MOVESTATE_ENABLE :
			PowerAxis1.Enable := TRUE;
			PowerAxis1.Enable_Positive := TRUE;
			PowerAxis1.Enable_Negative := TRUE;
			IF PowerAxis1.Status THEN
				state := MOVESTATE_FORWARD;
			ELSIF PowerAxis1.Error THEN
				state := MOVESTATE_ERROR;
			END_IF

		MOVESTATE_FORWARD :		(* start to first position *)
		MoveAxis1(
			axis := Axis1,
			Position := 63,	
			Velocity := 2,	
			Execute := TRUE
		);
		
		IF NOT MoveAxis1.Busy THEN
			MoveAxis1(axis := Axis1, Execute := FALSE);		// If axis is not busy, then execute move
			IF MoveAxis1.Error THEN
				state := MOVESTATE_ERROR;
			ELSE
				state := SEL(NOT bMove AND nIdlePosition = 1, MOVESTATE_NEWTARGETPOSITION, MOVESTATE_IDLE);
			(*If bMove=false and nIdlePosition=1, Movestate Idle, else NEWTARGETPOSITION*)
			END_IF
		END_IF

		MOVESTATE_NEWTARGETPOSITION :		(* change target position while moving *)
			MoveAxis1(
			axis := Axis1,
			Position := 55,	
			Velocity := 2,	
			Execute := TRUE
		);
		
		IF NOT MoveAxis1.Busy THEN
			MoveAxis1(axis := Axis1, Execute := FALSE);
			IF MoveAxis1.Error THEN
				state := MOVESTATE_ERROR;
			ELSE
				state := SEL(NOT bMove AND nIdlePosition = 2, MOVESTATE_FORWARD, MOVESTATE_IDLE);
				(*If bMove=FALSE && nIdlePosition=2 then MOVESTATE_IDLE; else MOVESTATE_FORWARD*)
			END_IF
		END_IF

		MOVESTATE_IDLE:
			HaltAxis1(axis := Axis1);
			
// 				IF bMove THEN
// 					state := MOVESTATE_NEWTARGETPOSITION;
// 		// 			HaltAxis1(axis := Axis1);	
// 				END_IF
				
		MOVESTATE_ERROR :
			state := SEL(Axis1.Status.Error, MOVESTATE_INIT, MOVESTATE_RESET);

		MOVESTATE_RESET :
// 			Reset.Execute := TRUE;
// 			IF Reset.Done THEN
// 				state := MOVESTATE_INIT;
// 			ELSIF Reset.Error THEN
// 				state := MOVESTATE_INIT; (* can't do anything here *)
// 			END_IF
			Reset.Execute := TRUE;
			state := MOVESTATE_INIT;

	END_CASE
	
PowerAxis1(axis := Axis1);
Reset(axis := Axis1);
// 
// 	fbMotor.EnablePower();	(* call the power function block *)
// 	fbMotor.MotorDosingPosition();	(* call the move function block *)
// 	fbMotor.MotorLoadingPosition();	(* call the reset function block *)
END_METHOD

METHOD MotorMove : BOOL
VAR_INPUT
	bMove : BOOL;
	nIdlePosition : INT; // 1: 63, 2: 70
	


END_VAR

VAR
	bLoadingPosition	: BOOL := process_gvl.fRobotInput.General_Bits.GPBitIN_15;
	bDosingPosition	: BOOL := process_gvl.fRobotInput.General_Bits.GPBitIN_16;
	trLoad      : R_TRIG;   // edge on bit 15
	trDose   	: R_TRIG;	// edge on bit 16
    bExecIssued : BOOL;     // latched once Busy=TRUE
END_VAR
IF nIdlePosition < 1 OR nIdlePosition > 2 THEN		// Rejects other Position values
	nIdlePosition := 1;
END_IF

Axis1();

CASE state OF
	MOVESTATE_INIT :	(* initialisation *)
		MoveAxis1.Execute := FALSE;
		Reset.Execute := FALSE;
		state := MOVESTATE_ENABLE;

	MOVESTATE_ENABLE :
		PowerAxis1.Enable := TRUE;
		PowerAxis1.Enable_Positive := TRUE;
		PowerAxis1.Enable_Negative := TRUE;
		IF PowerAxis1.Status THEN
// 			state := MOVESTATE_FORWARD;
			state := MOVESTATE_IDLE;
		ELSIF PowerAxis1.Error THEN
			state := MOVESTATE_ERROR;
		END_IF
		
	MOVESTATE_IDLE:		
		trLoad(CLK := process_gvl.fRobotInput.General_Bits.GPBitIN_15<>0);
		trDose(CLK := process_gvl.fRobotInput.General_Bits.GPBitIN_16<>0);
		
		IF trLoad.Q THEN
			state := MOVESTATE_FORWARD;
			bExecIssued := FALSE;   // prepare new command
		ELSIF trDose.Q THEN
			state := MOVESTATE_NEWTARGETPOSITION;
			bExecIssued := FALSE;
		ELSE
			state := MOVESTATE_IDLE;
		END_IF
		
	MOVESTATE_FORWARD :		(* start to first position *)        
		MoveAxis1(
			axis := Axis1,
			Position := 58,	
			Velocity := 2,	
			Execute := TRUE
		);
		IF NOT bExecIssued THEN
		// Present Execute until the FB acknowledges (Busy=TRUE once)
		MoveAxis1(axis := Axis1, Execute := FALSE); // If axis is not busy, then execute move  
		IF NOT MoveAxis1.Busy THEN 
				bExecIssued := TRUE;     // command has started
		END_IF 
		ELSE
			 // After start, keep calling with Execute FALSE
			 MoveAxis1(Axis := Axis1, Execute := FALSE);
		END_IF
		IF MoveAxis1.Error THEN 
			state := MOVESTATE_ERROR; 
		ELSIF bExecIssued AND NOT MoveAxis1.Busy THEN
			// Finished successfully → choose next
			bExecIssued := FALSE;
			state := SEL(bMove, MOVESTATE_NEWTARGETPOSITION, MOVESTATE_IDLE);
		END_IF
		
	MOVESTATE_NEWTARGETPOSITION : // IDLE POS 2
	MoveAxis1(
			axis := Axis1,
			Position := 63,	
			Velocity := 2,	
			Execute := TRUE
		);
		IF NOT bExecIssued THEN 
			MoveAxis1(
				axis := Axis1, Execute := FALSE);
			IF NOT MoveAxis1.Busy THEN 
				bExecIssued := TRUE;
			END_IF
		ELSE
			MoveAxis1(Axis := Axis1, Execute := FALSE);	
		END_IF
		IF MoveAxis1.Error THEN 
			state := MOVESTATE_ERROR; 
		ELSIF  bExecIssued AND NOT MoveAxis1.Busy THEN
			bExecIssued := FALSE;
			state := SEL(bMove, MOVESTATE_FORWARD, MOVESTATE_IDLE);
		END_IF 		

	MOVESTATE_ERROR :
		state := SEL(Axis1.Status.Error, MOVESTATE_INIT, MOVESTATE_RESET);

	MOVESTATE_RESET :
		Reset.Execute := TRUE;
		state := MOVESTATE_INIT;
END_CASE
	
PowerAxis1(axis := Axis1);
Reset(axis := Axis1);
END_METHOD

END_FUNCTION_BLOCK

// ---- POUs/Modules/FB_SolidSamplingModule.TcPOU
FUNCTION_BLOCK FB_SolidSamplingModule
VAR_INPUT
END_VAR
VAR_OUTPUT
END_VAR
VAR
END_VAR

END_FUNCTION_BLOCK

// ---- POUs/FB_Camera.TcPOU
FUNCTION_BLOCK FB_Camera
VAR_INPUT
	pRobot : POINTER TO FB_Robot;
END_VAR
VAR_OUTPUT
END_VAR
VAR
	    // Camera control
//     fbCam        :  FB_VN_SimpleCameraControl;
    eState       : ETcVnCameraState;
    hr           : HRESULT;

    // Software trigger (toggle TRUE → FALSE to grab one frame)
    bSoftTrig    : BOOL := FALSE;
    rSoftTrig    : R_TRIG;
    bPending     : BOOL := FALSE;

    // Images
    ipImageRaw   : ITcVnImage;               // raw from camera (Bayer GR8)
    ipImageGray  : ITcVnImage;               // grayscale after conversion
    ipImageRGB   : ITcVnImage;               // RGB canvas to draw on
    ipImageDisp  : ITcVnDisplayableImage;    // display handle for ADS
	ipImageDisp1 : ITcVnDisplayableImage;
// 	ipImageDispUndis : ITcVnDisplayableImage;
    // QR results
    ipDecoded    : ITcVnContainer;           // decoded data list
    ipContours   : ITcVnContainer;           // contours (for drawing)
    sQRCode      : STRING(255);

    // Drawing
    aRed         : TcVnVector4_LREAL := [0, 0, 255, 255];  // BGRA red
    font         : ETcVnFontType := TCVN_FT_HERSHEY_PLAIN;
	  clrRed			: TcVnVector4_LREAL := [255,0,0,255];
    clrBlue			: TcVnVector4_LREAL := [0,0,255,255];
	ipContour: ITcVnContainer;
	GetElementNum: INT;
	nPts: ULINT;
	nBufferSize: ULINT;

	ptTop: TcVnPoint2_LREAL;
	ptRight: TcVnPoint2_LREAL;
	ptLeft: TcVnPoint2_LREAL;
	ptBottom: TcVnPoint2_LREAL;

	// Camera calibration results
	
	fbCam				  :   FB_VN_GevCameraControl;
	aCameraMatrix             :   TcVnMatrix3x3_LREAL;
	aDistortionCoefficients   :   TcVnArray8_LREAL;
	aRotationMatrix           :   TcVnMatrix3x3_LREAL;
	aTranslationVector        :   TcVnVector3_LREAL;
	bInit: BOOL := TRUE;
	aCoordinatesWorld		:	ARRAY[0..4] OF TcVnPoint3_LREAL;
	aCoordinatesImage		:	ARRAY[0..4] OF TcVnPoint2_LREAL;
	ipImageRes: ITcVnImage;
	
	// QR code Dictionary lookup variables
	// ring buffer for last 8 QR numbers
    aQrIds      : ARRAY[0..7] OF DINT;   // filled FIFO-style
    iQrWrite    : INT := 0;              // next write index (0..7)
    nQrCount    : INT := 0;              // Nr of valid items (0..8)
    idQr        : DINT;                  // parsed numeric QR id (from sQRCode)
    bNewQrPulse : BOOL;                  // one-scan pulse when we store a new id
	
	  // Pose result of the QR (object pose in camera coordinates)
    aTagR       : TcVnMatrix3x3_LREAL;   // rotation matrix (QR->camera)
    aTagT       : TcVnVector3_LREAL;     // translation vector (mm; QR->camera)
	rv   		: TcVnVector3_LREAL;
    // convenience: latches
    bHavePose   : BOOL;
	
	 // --- one-shot control
    bRunOnce    : BOOL := FALSE;    // toggle TRUE for one cycle to run the test
    bBusy       : BOOL := FALSE;
	
    // (optional) GP mapping guard
    bParsedOk   : BOOL;
	
	fQrSizeMM   : LREAL := 23.0;         // <<< set your QR edge length (mm)
    aPts3D      : ARRAY[0..3] OF TcVnPoint3_LREAL;   // model points (QR frame)
    aPts2D      : ARRAY[0..3] OF TcVnPoint2_LREAL;   // image points (pixels)
    ipObjPts    : ITcVnContainer;        // vector<TcVnPoint3_LREAL>
    ipImgPts    : ITcVnContainer;        // vector<TcVnPoint2_LREAL>
	
	ipObjectPoints : ITcVnContainer;   // vector<TcVnPoint3_LREAL>  (3D model points)
    ipImagePoints  : ITcVnContainer;   // vector<TcVnPoint2_LREAL>  (2D image points)
	bReprojError  : LREAL;

    // --- Intrinsics (we try to read them; else we synthesize)
    aK              : TcVnMatrix3x3_LREAL;         // camera matrix
//     aDist80          : TcVnArray8_LREAL := [0,0,0,0,0,0,0,0]; // distortion zeroed for the synthetic test
	aDist80      : ARRAY[0..7] OF LREAL;   // zeros by default
    // --- SolvePnP outputs
    aR              : TcVnMatrix3x3_LREAL;
    aTt             : TcVnVector3_LREAL;
    bSolved         : BOOL;
	
	    // 2D/3D points (REAL versions!)
    aPts2D_R : ARRAY[0..3] OF TcVnPoint2_REAL;
    aPts3D_R : ARRAY[0..3] OF TcVnPoint3_REAL;
	    // --- containers (must be REAL types per Exp signature)
    ipRefPts    : ITcVnContainer;   // vector<TcVnPoint3_REAL>
	bCalibReady     : BOOL := FALSE;
	
	fbMakeT : FB_CreateTransformationMat;
	fbMakeT_1 : FB_CreateTransformationMat;
//     R_matrix       : TcVnMatrix3x3_LREAL;
//     t_matrix       : TcVnVector3_LREAL;
    T4x4_matrix       : TcVnMatrix;
	T4x4_matrix_1	  : TcVnMatrix;
	T4x4_matrix_result	  : TcVnMatrix;
	fbConvert : FB_MatConversion;
	fbRob : FB_Robot;
	fbMultiplyMat		: FB_MultiplyMatrices4x4;
	
END_VAR
	
VAR_OUTPUT
	_pose : ST_PoseLREAL;
END_VAR

PROPERTY Pose : REFERENCE TO ST_PoseLREAL // Property to obtain pose of Tag w.r.t. camera
GET
Pose REF= _pose;
END_GET
SET
END_SET
END_PROPERTY

METHOD QRCodefinal : BOOL
VAR_INPUT
END_VAR

VAR
END_VAR

VAR_OUTPUT
END_VAR
// --- Provider state machine ---
eState := fbCam.GetState();

CASE eState OF
    TCVN_CS_ERROR:
        hr := fbCam.Reset();

    TCVN_CS_INITIAL, TCVN_CS_INITIALIZING, TCVN_CS_INITIALIZED,
    TCVN_CS_OPENING, TCVN_CS_OPENED, TCVN_CS_STARTACQUISITION:
        hr := fbCam.StartAcquisition();
END_CASE

// --- Read calibration once, when ACQUIRING ---
IF (eState = TCVN_CS_ACQUIRING) AND NOT bCalibReady THEN
    hr := fbCam.GetCameraMatrix(aCameraMatrix);
    IF SUCCEEDED(hr) THEN
        hr := fbCam.GetDistortionCoefficients(aDistortionCoefficients);  // length must match your calibration
    END_IF
    bCalibReady := SUCCEEDED(hr);
END_IF

// --- Work only when ACQUIRING ---
IF eState = TCVN_CS_ACQUIRING THEN

    // Software trigger (edge)
    rSoftTrig(CLK := bSoftTrig);
    IF rSoftTrig.Q THEN
        hr := fbCam.TriggerImage();
        bPending := TRUE;
    END_IF

    // One-shot trigger support (optional)
    IF bRunOnce AND NOT bBusy THEN
        bBusy := TRUE;
        hr := fbCam.TriggerImage();
        bPending := TRUE;
    END_IF

    IF bPending THEN
        hr := fbCam.GetCurrentImage(ipImageRaw);

        IF SUCCEEDED(hr) AND (ipImageRaw <> 0) THEN
            // 1) RAW (Bayer GR8) -> GRAY
            hr := F_VN_ConvertColorSpace(
                    ipSrcImage := ipImageRaw,
                    ipDestImage := ipImageGray,
                    eTransform := TCVN_CST_BAYER_GR_TO_GRAY,
                    hrPrev := hr);

            // 2) QR decode (+ contours)
            hr := F_VN_ReadQRCodeExp(
                    ipSrcImage      := ipImageGray,
                    ipDecodedData   := ipDecoded,
                    ipContours      := ipContours,
                    nCodeNumber     := 1,
                    eSearchStrategy := TCVN_CSS_ONLY_NOT_INVERTED + TCVN_CSS_ONLY_NOT_FLIPPED,
                    hrPrev          := hr);

            // 3) Prepare RGB canvas if something was found
            IF (ipDecoded <> 0) AND (ipContours <> 0) THEN
                hr := F_VN_ConvertColorSpace(
                        ipSrcImage := ipImageGray,
                        ipDestImage := ipImageRGB,
                        eTransform := TCVN_CST_GRAY_TO_RGB,
                        hrPrev := hr);
            END_IF

            // 4) If decoded, export text, draw contour, store ID
            IF SUCCEEDED(hr) AND (ipDecoded <> 0) THEN
                hr := F_VN_ExportSubContainer_String(
                        ipContainer := ipDecoded,
                        nIndex := 0,
                        sText := sQRCode,
                        nMaxLength := SIZEOF(sQRCode)-1,
                        hrPrev := hr);

                IF SUCCEEDED(hr) AND (ipContours <> 0) THEN
                    hr := F_VN_DrawContours(ipContours, -1, ipImageRGB, clrRed, 3, hr);
                END_IF

                // push into ring buffer (no validation here; add if needed)
                idQr := STRING_TO_DINT(sQRCode);
                aQrIds[iQrWrite] := idQr;
                iQrWrite := (iQrWrite + 1) MOD 8;
                IF nQrCount < 8 THEN nQrCount := nQrCount + 1; END_IF
            END_IF

            // 5) Extract QR corner points (TL, TR, BR, BL)
            IF (ipContours <> 0) THEN
                ipContour := 0;
                hr := F_VN_GetAt_ITcVnContainer(ipContours, ipContour, 0, hr);

                IF (ipContour <> 0) THEN
                    ipContour.GetElementNum(nPts);

                    IF nPts > 0 THEN
                        // Extremes → TL, TR, BR, BL
                        hr := F_VN_ContourExtremePoint(ipContour:=ipContour, eDirection:=TCVN_EPD_TOP_LEFT,     aExtremePoint:=ptTop,    hrPrev:=S_OK);
                        hr := F_VN_ContourExtremePoint(ipContour:=ipContour, eDirection:=TCVN_EPD_RIGHT_TOP,    aExtremePoint:=ptRight,  hrPrev:=hr);
                        hr := F_VN_ContourExtremePoint(ipContour:=ipContour, eDirection:=TCVN_EPD_BOTTOM_RIGHT, aExtremePoint:=ptBottom, hrPrev:=hr);
                        hr := F_VN_ContourExtremePoint(ipContour:=ipContour, eDirection:=TCVN_EPD_LEFT_BOTTOM,  aExtremePoint:=ptLeft,   hrPrev:=hr);

                        IF SUCCEEDED(hr) THEN
                            // draw corner marks
                            hr := F_VN_DrawPointExp(TO_UDINT(ptTop[0]),    TO_UDINT(ptTop[1]),    ipImageRGB, TCVN_DS_PLUS, clrBlue, 5, -1, TCVN_LT_4_CONNECTED, hr);
                            hr := F_VN_DrawPointExp(TO_UDINT(ptRight[0]),  TO_UDINT(ptRight[1]),  ipImageRGB, TCVN_DS_PLUS, clrBlue, 5, -1, TCVN_LT_4_CONNECTED, hr);
                            hr := F_VN_DrawPointExp(TO_UDINT(ptBottom[0]), TO_UDINT(ptBottom[1]), ipImageRGB, TCVN_DS_PLUS, clrBlue, 5, -1, TCVN_LT_4_CONNECTED, hr);
                            hr := F_VN_DrawPointExp(TO_UDINT(ptLeft[0]),   TO_UDINT(ptLeft[1]),   ipImageRGB, TCVN_DS_PLUS, clrBlue, 5, -1, TCVN_LT_4_CONNECTED, hr);

                            // --- Build 3D model (REAL) TL,TR,BR,BL (Z=0 plane) ---
                            aPts3D_R[0][0] := LREAL_TO_REAL(-fQrSizeMM*0.5);  aPts3D_R[0][1] := LREAL_TO_REAL(-fQrSizeMM*0.5);  aPts3D_R[0][2] := 0.0;
                            aPts3D_R[1][0] := LREAL_TO_REAL( fQrSizeMM*0.5);  aPts3D_R[1][1] := LREAL_TO_REAL(-fQrSizeMM*0.5);  aPts3D_R[1][2] := 0.0;
                            aPts3D_R[2][0] := LREAL_TO_REAL( fQrSizeMM*0.5);  aPts3D_R[2][1] := LREAL_TO_REAL( fQrSizeMM*0.5);  aPts3D_R[2][2] := 0.0;
                            aPts3D_R[3][0] := LREAL_TO_REAL(-fQrSizeMM*0.5);  aPts3D_R[3][1] := LREAL_TO_REAL( fQrSizeMM*0.5);  aPts3D_R[3][2] := 0.0;

                            // --- 2D image points (REAL) in the same order ---
                            aPts2D_R[0][0] := LREAL_TO_REAL(ptTop[0]);    aPts2D_R[0][1] := LREAL_TO_REAL(ptTop[1]);
                            aPts2D_R[1][0] := LREAL_TO_REAL(ptRight[0]);  aPts2D_R[1][1] := LREAL_TO_REAL(ptRight[1]);
                            aPts2D_R[2][0] := LREAL_TO_REAL(ptBottom[0]); aPts2D_R[2][1] := LREAL_TO_REAL(ptBottom[1]);
                            aPts2D_R[3][0] := LREAL_TO_REAL(ptLeft[0]);   aPts2D_R[3][1] := LREAL_TO_REAL(ptLeft[1]);

                            // --- Create REAL containers and fill ---
                            ipRefPts := 0; ipImgPts := 0;
                            hr := F_VN_CreateContainer(ipRefPts, ContainerType_Vector_TcVnPoint3_REAL, 4, hr);
                            IF SUCCEEDED(hr) THEN
                                hr := F_VN_CreateContainer(ipImgPts, ContainerType_Vector_TcVnPoint2_REAL, 4, hr);
                            END_IF

                            IF SUCCEEDED(hr) THEN
                                hr := F_VN_SetAt_TcVnPoint3_REAL(aPts3D_R[0], ipRefPts, 0, hr);
                                hr := F_VN_SetAt_TcVnPoint3_REAL(aPts3D_R[1], ipRefPts, 1, hr);
                                hr := F_VN_SetAt_TcVnPoint3_REAL(aPts3D_R[2], ipRefPts, 2, hr);
                                hr := F_VN_SetAt_TcVnPoint3_REAL(aPts3D_R[3], ipRefPts, 3, hr);

                                hr := F_VN_SetAt_TcVnPoint2_REAL(aPts2D_R[0], ipImgPts, 0, hr);
                                hr := F_VN_SetAt_TcVnPoint2_REAL(aPts2D_R[1], ipImgPts, 1, hr);
                                hr := F_VN_SetAt_TcVnPoint2_REAL(aPts2D_R[2], ipImgPts, 2, hr);
                                hr := F_VN_SetAt_TcVnPoint2_REAL(aPts2D_R[3], ipImgPts, 3, hr);
                            END_IF

                            // --- SolvePnP (Exp) → full 6D pose ---
                            bHavePose := FALSE;
                            IF SUCCEEDED(hr) AND bCalibReady THEN
                                hr := F_VN_SolvePnPExp(
                                        ipImagePoints           := ipImgPts,
                                        ipReferencePoints       := ipRefPts,
                                        aCameraMatrix           := aCameraMatrix,
                                        aDistortionCoefficients := aDistortionCoefficients, // exact length!
                                        aRotationMatrix         := aTagR,
                                        aTranslationVector      := aTagT,
                                        fReprojError            := bReprojError,
                                        eMethod                 := TCVN_SPM_ITERATIVE,      // your build
                                        bUseExtrinsicGuess      := FALSE,
                                        hrPrev                  := hr);

                                bHavePose := SUCCEEDED(hr);
								
								IF bHavePose THEN
									rv := fbConvert.RmatToRotVec(aTagR);
									// Create Transformation matrix using aTagR and aTagT.
								 	_pose.R_Mat := aTagR; //Rotation matrix
									_pose.T_Mat := aTagT; //Translation matrix
									
									fbMakeT.R_mat := _pose.R_Mat;
									fbMakeT.t_mat := _pose.T_Mat;
									fbMakeT();
									// outputs a valid TcVnMatrix pointing to internal 4x4 LREALs
									T4x4_matrix := fbMakeT.Tx_mat;				
// 									T4x4_matrix_1:=fbRob.RobotPose();  // error
									
									fbRob.RobotPose();				
									_pose.R_Mat := fbRob.r1_matrix;
									_pose.T_Mat := fbRob.v1_matrix;

									fbMakeT_1.R_mat := _pose.R_Mat;
									fbMakeT_1.t_mat := _pose.T_Mat;
									fbMakeT_1();
									
									T4x4_matrix_1:= fbMakeT_1.Tx_mat;
									
(*Multiply cam_T_qr to base_T_tcp*)
									fbMultiplyMat(M1:=T4x4_matrix, M2:=T4x4_matrix_1);	 
									T4x4_matrix_result := fbMultiplyMat.M_result;
(*Multiply xx_T_xx to xx_T_xx*)
									process_gvl.fRobotOutput.General_Register1.Floats.Floats[3] := LREAL_TO_REAL(aTagT[0]);
									process_gvl.fRobotOutput.General_Register1.Floats.Floats[4] := LREAL_TO_REAL(aTagT[1]);
									process_gvl.fRobotOutput.General_Register1.Floats.Floats[5] := LREAL_TO_REAL(aTagT[2]);
									process_gvl.fRobotOutput.General_Register1.Floats.Floats[0] := LREAL_TO_REAL(rv[0]);
									process_gvl.fRobotOutput.General_Register1.Floats.Floats[1] := LREAL_TO_REAL(rv[1]);
									process_gvl.fRobotOutput.General_Register1.Floats.Floats[2] := LREAL_TO_REAL(rv[2]);
									
								END_IF
                            END_IF

                            // tidy temp containers
                            ipRefPts := 0; ipImgPts := 0;
                        END_IF
                    END_IF
                END_IF
            END_IF

            // 6) Show in ADS Image Watch
            hr := F_VN_CopyIntoDisplayableImage(ipSrcImage:= ipImageRGB, ipDestImage:=ipImageDisp1, hr );
            hr := F_VN_TransformIntoDisplayableImage(ipImageRGB, ipImageDisp, hr);

            // cleanup for next trigger
            ipDecoded    := 0;
            ipContours   := 0;
            ipImageRaw   := 0;
            ipImageGray  := 0;
            ipImageRGB   := 0;
            bPending     := FALSE;
        END_IF
    END_IF
END_IF

// allow one-shot retrigger
IF NOT bRunOnce THEN
    bBusy := FALSE;
END_IF
END_METHOD

END_FUNCTION_BLOCK

// ---- POUs/FB_MultiplyMatrices4x4.TcPOU
FUNCTION_BLOCK FB_MultiplyMatrices4x4
VAR_INPUT
	M1 : TcVnMatrix;
	M2 : TcVnMatrix;
	hr : HRESULT :=S_OK;
END_VAR
VAR_OUTPUT
	M_result : TcVnMatrix;
END_VAR
VAR
END_VAR



hr := F_VN_MultiplyMatrices(stSrcMatrix1 := M1, stSrcMatrix2 := M2, hrPrev := S_OK, stDestMatrix := M_result);

END_FUNCTION_BLOCK

// ---- POUs/FB_LoadCell.TcPOU
FUNCTION_BLOCK FB_LoadCell EXTENDS FB_SolidSamplingModule
VAR_INPUT
END_VAR
VAR_OUTPUT
END_VAR
VAR
END_VAR

END_FUNCTION_BLOCK

// ---- POUs/FB_MagStirrer.TcPOU
FUNCTION_BLOCK FB_MagStirrer EXTENDS FB_Tools
VAR_IN_OUT
	RxBufferEL : ComBuffer; (* Receive data buffer; used with all receive function blocks *)
    TxBufferEL : ComBuffer; (* Transmit data buffer; used with all receive function blocks *)
END_VAR
VAR
	
	
	stIn_EL6001 AT %I*     : EL6inData22B; (* linked to the EL6001 in the TwinCAT System Manager *)
    stOut_EL6001 AT %Q*    : EL6outData22B;(* linked to the EL6001 in the TwinCAT System Manager *)
	fbEL6001Ctrl       : SerialLineControl;
    bEL6001CtrlError   : BOOL;
    eEL6001CtrlErrorID : ComError_t;
END_VAR

fbEL6001Ctrl(
    Mode:= SERIALLINEMODE_EL6_22B, 
    pComIn:= ADR(stIn_EL6001), 
    pComOut:= ADR(stOut_EL6001), 
    SizeComIn:= SIZEOF(stIn_EL6001), 
    Error=> bEL6001CtrlError, 
    ErrorID=> eEL6001CtrlErrorID, 
    TxBuffer:= TxBufferEL, 
    RxBuffer:= RxBufferEL );

METHOD SetRPM : BOOL
VAR_INPUT
END_VAR
END_METHOD

METHOD TriggerStirrer : BOOL
VAR
// 	fbReceiveString	:	ReceiveString;
// 	fbSendString	:	SendString := 'start';
END_VAR
// SendString(SendString:= SentString,
// 			TxBuffer := TxBuffer);
// ReceiveString(Prefix := Prefix,
// 			Suffix := Suffix,
// 			Timeout	:= Timeout,
// 			Reset	:=	Reset,
// 			ReceivedString:= ReceivedString,
// 			RXbuffer := RXBuffer);
END_METHOD

END_FUNCTION_BLOCK

// ---- POUs/FB_PeristalticPump.TcPOU
FUNCTION_BLOCK FB_PeristalticPump EXTENDS FB_AnalyticalDevices
VAR_INPUT
END_VAR
VAR_OUTPUT
END_VAR
VAR
END_VAR

METHOD TriggerPumpOff : BOOL
VAR_INPUT
END_VAR
END_METHOD

METHOD TriggerPumpOn : BOOL
VAR_INPUT
END_VAR
END_METHOD

END_FUNCTION_BLOCK

// ---- POUs/FB_SerialCom.TcPOU
FUNCTION_BLOCK FB_SerialCom
VAR_IN_OUT
	TxBuffer	: ComBuffer;
	RxBuffer	: ComBuffer;
END_VAR
VAR
// 	Timer		: TON := (PT:=T#1S);
// 	fbSend		: SendData;
// 	bSendBusy	: BOOL;
// 	eSendErrorID: ComError_t;
// 
// 	fbReceive		: ReceiveData;
// 	sReceivedData	: STRING;
// 	sLastReceivedString: STRING;
// 	bStringReceived	: BOOL;
// 	bReceiveBusy	: BOOL;
// 	bReceiveError	: BOOL;
// 	eReceiveErrorID	: ComError_t;
// 	bReceiveTimeout	: BOOL;
// 	nReceiveCounter	: UDINT;
// 	
// 	aCmd        : ARRAY[0..6] OF STRING := ['s','t','a','r','t','\r','\n']; // "start"
// 	//47, 40, 95, 65, 41, 13, 10
// 	
// 	  pPrefix         : BYTE;
// 	  LenPrefix       : BYTE;
// 	  pSuffix         : BYTE;
// 	  LenSuffix       : BYTE;
// 	  pReceiveData    : BYTE;
// 	  SizeReceiveData : DINT;
// 	  Timeout         : TIME := T#1S;
// 	  Reset           : BOOL;
// 	  
// 	  sPrefix  : STRING(1) := '';              // no prefix, or STX if required
//       sSuffix  : STRING(1) := '';              // no suffix, or ETX if required
//       aReceive : ARRAY[0..255] OF STRING;

	SendString: STRING:= 'start';
	Busy : BOOL;
    Error: ComError_t;
	fbSendString : SendString;
	fbReceiveString : ReceiveString;
	Prefix : STRING:= '';
    Suffix : STRING := '';
    Timeout : TIME;
    Reset :BOOL;
	StringReceived: BOOL;
    RxTimeout : BOOL;
	ReceivedString : STRING;
END_VAR

// Call the send block every second to repeat the transmission.
// Also call the block as long as it is busy to finish a transmission.
// Timer(IN:=TRUE);
// IF Timer.Q OR fbSend.Busy THEN
// 	Timer(IN:=FALSE); (* reset timer *)
// 	fbSend(	pSendData := ADR(aCmd),
// 			Length:=SIZEOF(aCmd),
// 			TXbuffer:= TxBuffer,
// 			Busy=> bSendBusy,
// 			Error=> );
// 	IF fbSend.Error <> COMERROR_NOERROR THEN
// 		eSendErrorID := fbSend.Error;
// 	END_IF
// END_IF

// 	Receive STRING data:
// 	The block receives any data strings beginning with a STX ($02) and ending with an ETX ($03) character.	
// fbReceive(	pPrefix:=ADR(pPrefix),
// 		  	LenPrefix:=LenPrefix,
// 			pSuffix:=ADR(pSuffix),
// 			LenSuffix:=LenSuffix,
// 			pReceiveData:=ADR(pReceiveData),
// 			SizeReceiveData:=SIZEOF(pReceiveData),		
// 			Timeout:=Timeout,
// // 			Reset:=Reset
// 			RXbuffer:=RxBuffer);

// 	fbReceive(	pPrefix:= 0,
// 		  	LenPrefix:=0,
// 			pSuffix:=0,
// 			LenSuffix:=0,
// 			pReceiveData:=ADR(aReceive),
// 			SizeReceiveData:=SIZEOF(aReceive),		
// 			Timeout:=Timeout,
// // 			Reset:=Reset
// 			RXbuffer:=RxBuffer);
	
// IF fbReceive.Error <> COMERROR_NOERROR THEN
// 	eReceiveErrorID := fbReceive.Error;
// END_IF
// IF bStringReceived THEN
// 	nReceiveCounter := nReceiveCounter + 1;
// 	sLastReceivedString := sReceivedString;
// END_IF

fbSendString(SendString:= SendString, TXbuffer:=TXbuffer);
fbReceiveString(Prefix := Prefix, Suffix:= Suffix, Timeout:=Timeout, Reset:=Reset, ReceivedString:= ReceivedString, RXbuffer:=RXBuffer);

END_FUNCTION_BLOCK

// ---- POUs/FB_Test.TcPOU
FUNCTION_BLOCK FB_Test
VAR
    hr              :   HRESULT;
    ipImageIn       :   ITcVnImage;
    ipImageInDisp   :   ITcVnDisplayableImage;
    fbCameraControl :   FB_VN_SimpleCameraControl;
    eCameraState    :   ETcVnCameraState;
    nNewImageCounter:   UINT;
END_VAR

eCameraState := fbCameraControl.GetState();

// CameraControl is in error state, so try to reset the camera connection
IF eCameraState = TCVN_CS_ERROR THEN
    hr := fbCameraControl.Reset();

// Camera not yet streaming
ELSIF eCameraState < TCVN_CS_ACQUIRING THEN
    hr := fbCameraControl.StartAcquisition();

// Camera streaming
ELSIF eCameraState = TCVN_CS_ACQUIRING THEN
    hr := fbCameraControl.GetCurrentImage(ipImageIn);

    // Check if new Image was received
    IF SUCCEEDED(hr) AND ipImageIn <> 0 THEN
        nNewImageCounter := nNewImageCounter + 1;

        // Place to call vision algorithms
        hr := F_VN_TransformIntoDisplayableImage(ipImageIn, ipImageInDisp, hr);
    END_IF

END_IF

END_FUNCTION_BLOCK

// ---- POUs/Modules/FB_LoadingStationA.TcPOU
FUNCTION_BLOCK FB_LoadingStationA
VAR_INPUT
END_VAR
VAR_OUTPUT
END_VAR
VAR
END_VAR

END_FUNCTION_BLOCK

// ---- POUs/Modules/FB_StirringModule.TcPOU
FUNCTION_BLOCK FB_StirringModule
VAR_INPUT
END_VAR
VAR_OUTPUT
END_VAR
VAR
END_VAR

END_FUNCTION_BLOCK
